{attribute 'linkalways'} 
{attribute 'no_explicit_call' := 'This FB is a CLASS and must be accessed using methods or properties'}
{attribute 'enable_dynamic_creation'}
FUNCTION_BLOCK Node_F_VN_MultiplyImageWithScalar EXTENDS VisionNode
VAR
    fScalar : _LREAL(0.0);
    ipSrcImage : _ITcVnImage;
    ipDestImage : _ITcVnImage;
    hrPrev : _HRESULT(S_OK);
	hresult : _HRESULT(S_OK);
END_VAR

METHOD PUBLIC  Clone : I_Node
VAR
	pNode : POINTER TO Node_F_VN_MultiplyImageWithScalar;
END_VAR
pNode := __NEW(Node_F_VN_MultiplyImageWithScalar);
Clone := pNode^;
END_METHOD

METHOD FB_init : BOOL
VAR_INPUT
	bInitRetains : BOOL; // if TRUE, the retain variables are initialized (warm start / cold start)
	bInCopyCode : BOOL;  // if TRUE, the instance afterwards gets moved into the copy code (online change)
END_VAR
AddInput('fScalar', fScalar);
AddInput('ipSrcImage', ipSrcImage);
AddInput('hrPrev', hrPrev);
AddOutput('ipDestImage', ipDestImage);
AddOutput('hresult',hresult);
END_METHOD

METHOD PROTECTED OnExecute : HRESULT
hresult.Value := F_VN_MultiplyImageWithScalar(
    fScalar := fScalar.Value,
    ipSrcImage := ipSrcImage.Value,
	ipDestImage := ipDestImage.Value,
	hrPrev:= hrPrev.Value);
END_METHOD

METHOD PUBLIC PreExecutionCheck
VAR_INPUT
	Check : I_PreExecutionChecks;
END_VAR
IF FAILED(hrPrev.Value) THEN
    RETURN;
END_IF

Check.IsTrue(ipSrcImage.IsValid, 'ipSrcImage must contain an image');
END_METHOD

END_FUNCTION_BLOCK

(* stored: Version 1.1.0.1, ProductVersion 3.1.4024.13
   POU Node_F_VN_MultiplyImageWithScalar: Id {4569af38-c2f0-0a94-35f7-f0b5f1dd3f5b}, SpecialFunc None
   Folder Constructor: Id {bf8b3c2e-f5b0-0882-324e-9e79b0461fd9}
   Method Clone: Id {e4474127-2c57-0320-0ea0-29c1e8e832d0}
   Method FB_init: Id {08ea7bf3-3a91-069f-3a31-082228ff8d6a}
   Method OnExecute: Id {76d2a717-3207-032f-192e-8806cfa8cdfe}
   Method PreExecutionCheck: Id {98df4c08-2b93-0770-1bcd-87972c890a3a} *)
